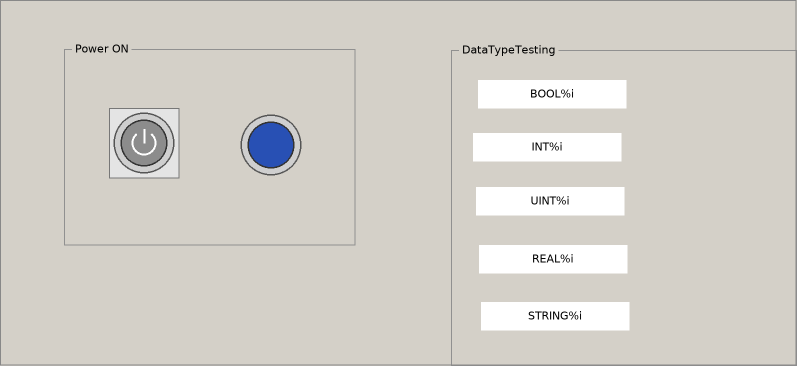
VISUALIZATION HMI  // 797x366
    GroupBox (64,41 291x204), "Power ON"
        PowerSwitch (45,67 70x70), variable: MAIN.bStart, behaviour: TOGGLE, style: Switch-PowerSwitch-Gray
        Lamp1 (172,69 70x70), variable: MAIN.bEnable, style: Lamp-Lamp1-Blue
    GroupBox (451,42 346x324), "DataTypeTesting"
        Textfield (26,37 150x30), "BOOL%i", text variable: MAIN.bEnable
        Textfield (21,90 150x30), "INT%i", text variable: MAIN.nINT
        Textfield (24,144 150x30), "UINT%i", text variable: MAIN.nUINT
        Textfield (27,202 150x30), "REAL%i", text variable: MAIN.fREAL
        Textfield (29,259 150x30), "STRING%i"
END_VISUALIZATION

(* stored: Version 1.1.0.1, ProductVersion 3.1.4024.12
   Visu HMI: Id {c7ee00a3-5f18-4b36-ba1e-9e8064ec0ee9} *)
